Staubli VAL3: remGetWorld.pgx

program remGetWorld(string& sReturn[] (dimensions=1))
  local point pHere
  local trsf trHere
begin
  // Return the world position values, ignoring the current frame.
  //
  logMsg("call remGetWorld")
  pHere=here(tSensorTool,world)
  trHere=pHere.trsf
  sReturn="GETWORLD"
  sReturn=sReturn+" "+toString(sNumConv,trHere.x)
  sReturn=sReturn+" "+toString(sNumConv,trHere.y)
  sReturn=sReturn+" "+toString(sNumConv,trHere.z)
  sReturn=sReturn+" "+toString(sNumConv,trHere.rx)
  sReturn=sReturn+" "+toString(sNumConv,trHere.ry)
  sReturn=sReturn+" "+toString(sNumConv,trHere.rz)
end
